PROGRAM DatenRangieren
VAR	
	VersionsText: STRING := 'Labor Linearachse V2.0';
END_VAR

VersionsInfo.Ver := MAXSTRING_TO_BYTEARR(VersionsText);

IF VersionsInfo.Befehle = 16#00 THEN	// lokale Ein- und Ausgänge verwenden
	SimDI.S1 := BitLesen(Plc_dSub.DI_LowByte,0);
	
	Plc_dSub.DQ_LowByte := AlleBitSetzen(	SimDa.P1,
											FALSE,
											FALSE,
											FALSE,
											FALSE,	
											FALSE,	
											FALSE,										
											FALSE);	
ELSE	// Simulation (Digital Twin) verwenden
	SimDI.S1 := BitLesen(DigInput.DI[0],0);
	
	DigOutput.DA[0] := AlleBitSetzen(	SimDa.P1,
										FALSE,
										FALSE,
										FALSE,
										FALSE,	
										FALSE,	
										FALSE,										
										FALSE);	
END_IF

END_PROGRAM

(* stored: Version 1.1.0.1, ProductVersion 3.1.4024.4
   POU DatenRangieren: Id {ad49a684-d9e6-4dba-bece-08745f191ac1}, SpecialFunc None *)
